// TIA Portal V21 export
TYPE "Rcp_VacuumFiller"
   STRUCT
      SelezTipoProdotto : Bool;   // 0=Olio / 1=Salamoia
      VelocitàPompaRiscladamentoOlio : Real;
      TemperaturaRiscaldamentoOlio : Real;   // Temperatura richiesta riscaldamento olio
      TemperaturaMinRiscaldamentoOlio : Real;   // Temperatura minima riscaldamento olio
      TemperaturaMaxRiscaldamentoOlio : Real;   // Temperatura massima riscaldamento olio
      TemperaturaHystRiscaldamentoOlio : Real;   // Temperatura isteresi riscaldamento olio
      VelocitàPompaRiscladamentoSalamoia : Real;
      TemperaturaRiscaldamentoSalamoia : Real;   // Temperatura richiesta riscaldamento salamoia
      TemperaturaMinRiscaldamentoSalamoia : Real;   // Temperatura minima riscaldamento salamoia
      TemperaturaMaxRiscaldamentoSalamoia : Real;   // Temperatura massima riscaldamento salamoia
      TemperaturaHystRiscaldamentoSalamoia : Real;   // Temperatura isteresi riscaldamento salamoia
   END_STRUCT;
END_TYPE
